FUNCTION_BLOCK FB_MovingHeadOnCommand IMPLEMENTS I_Command
VAR
	refMovingHead : REFERENCE TO FB_MovingHead;
END_VAR

METHOD Execute
IF (__ISVALIDREF(THIS^.refMovingHead)) THEN
	THIS^.refMovingHead.On();
END_IF
END_METHOD

METHOD FB_init : BOOL
VAR_INPUT
	bInitRetains 	: BOOL; // if TRUE, the retain variables are initialized (warm start / cold start)
	bInCopyCode 	: BOOL;  // if TRUE, the instance afterwards gets moved into the copy code (online change)
	refMovingHead 	: REFERENCE TO FB_MovingHead;
END_VAR
IF (__ISVALIDREF(refMovingHead)) THEN
	THIS^.refMovingHead REF= refMovingHead;
ELSE
	THIS^.refMovingHead REF= 0;
END_IF
END_METHOD

END_FUNCTION_BLOCK

(* stored: Version 1.1.0.1, ProductVersion 3.1.4022.18
   POU FB_MovingHeadOnCommand: Id {7968216d-3548-4918-ac22-4f07e36a3613}, SpecialFunc None
   Method Execute: Id {e6940612-6cee-412d-b5ae-daf79e7ef8f5}
   Method FB_init: Id {c2540567-b370-44c2-869d-0602404cfd87} *)
